// TIA Portal V17 export
FUNCTION "FC_风机燃气控制" : Void   // FC, LAD
{ S7_Optimized_Access := 'TRUE' }
   VAR_TEMP
      风机控制输出值 : Real;
      风压过渡 : Int;
   END_VAR
BEGIN

REGION Network 1: 风机运行控制
   // 常开触点风机运行按与常闭触点风机故障反馈串联，当风机运行按接通且风机故障反馈未动作时，驱动风机运行线圈Q4.4
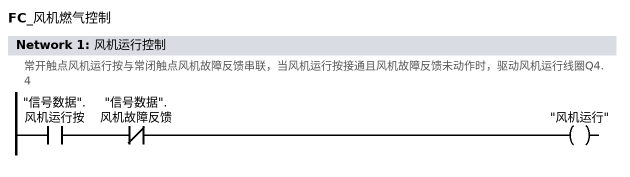
   RUNG wire#powerrail
      Contact( "信号数据".风机运行按 )
      I_Contact( "信号数据".风机故障反馈 )
      Coil( "风机运行" )
   END_RUNG
   // the same network as SCL:
   "风机运行" := "信号数据".风机运行按 AND NOT "信号数据".风机故障反馈;
END_REGION
END_FUNCTION
